PROGRAM MAIN
VAR_INPUT
	// Nostimen tulot
	iElevatorSensor AT %IX1.0: BOOL; // nostimen valoanturi
	iElevatorIsLifted AT %IX1.1: BOOL; // nostin on ajettu ylärajalle
	iElevatorIsDescended AT %IX1.2: BOOL; // nostin on ajettu alarajalle
	iElevatorConveyorRunning AT %IX1.3: BOOL; // nostimen kuljetin pyörii
	
	// Kuljetin 2 tulot
	iConveyor2Sensor AT %IX2.0: BOOL; // Valokenno kuljetin 2 ennen työnnintä
	iPusherPushed AT %IX2.1: BOOL; // Työnnnin on ulkona
	iPusherRetracted AT %IX2.2: BOOL; // Työnnin on sisällä
	iConveyor2Running AT %IX2.3: BOOL; // kuljetin 2 pyörii
	
	// Kuljetin 1 tulot
	iConveyor1Running AT %IX3.0: BOOL; // Kuljetin 1 pyörii
END_VAR

VAR_OUTPUT
	// Kuljetin 1 lähdöt
	qConveyor1 AT %QX0.0: BOOL; // Kuljetin 1 ajo
	
	// Nostimen lähdöt
	qElevatorConveyor AT %QX1.0: BOOL; // Nostimen kuljetin ajo
	qElevatorUp AT %QX1.1: BOOL; // Nostimen nosto ylös
	qElevatorDown AT %QX1.2: BOOL; // Nostimen lasku alas
	
	// Kuljetin 2 lähdöt
	qConveyor2 AT %QX2.0: BOOL; // Kuljetin 2 ajo 
	qPusherPush AT %QX2.1: BOOL; // Työnnin eteen
	qPusherRetract AT %QX2.2: BOOL; // Työnnin taakse
	
	// Laatikon lähtö 
	qBoxShaker AT %QX3.0: BOOL; // Laatikon tärytin
END_VAR

VAR
	ManConveyor1: BOOL; // Kuljetin 1 ajo
	ManElevatorConveyor: BOOL; // Nostimen kuljetin ajo
	ManElevatorUp: BOOL; // Nostimen nosto ylös
	ManElevatorDown: BOOL; // Nostimen lasku alas
	ManConveyor2: BOOL; // Kuljetin 2 ajo 
	ManPusherPush: BOOL; // Työnnin eteen
	ManPusherRetract: BOOL; // Työnnin taakse
	ManBoxShaker: BOOL; // Laatikon tärytin	
	Manual_mode: BOOL;
	Auto_mode: BOOL;
	Lamp: BOOL;
	START: BOOL;
	Seq1: BOOL;
	Seq2: BOOL;
	Seq3: BOOL;
	Seq4: BOOL;
	Seq5: BOOL;
	STOP: BOOL;
END_VAR
VAR // added by the converter: edge detectors and wires of the graphical bodies
    _ft1 : F_TRIG;
    _w1 : BOOL;
END_VAR

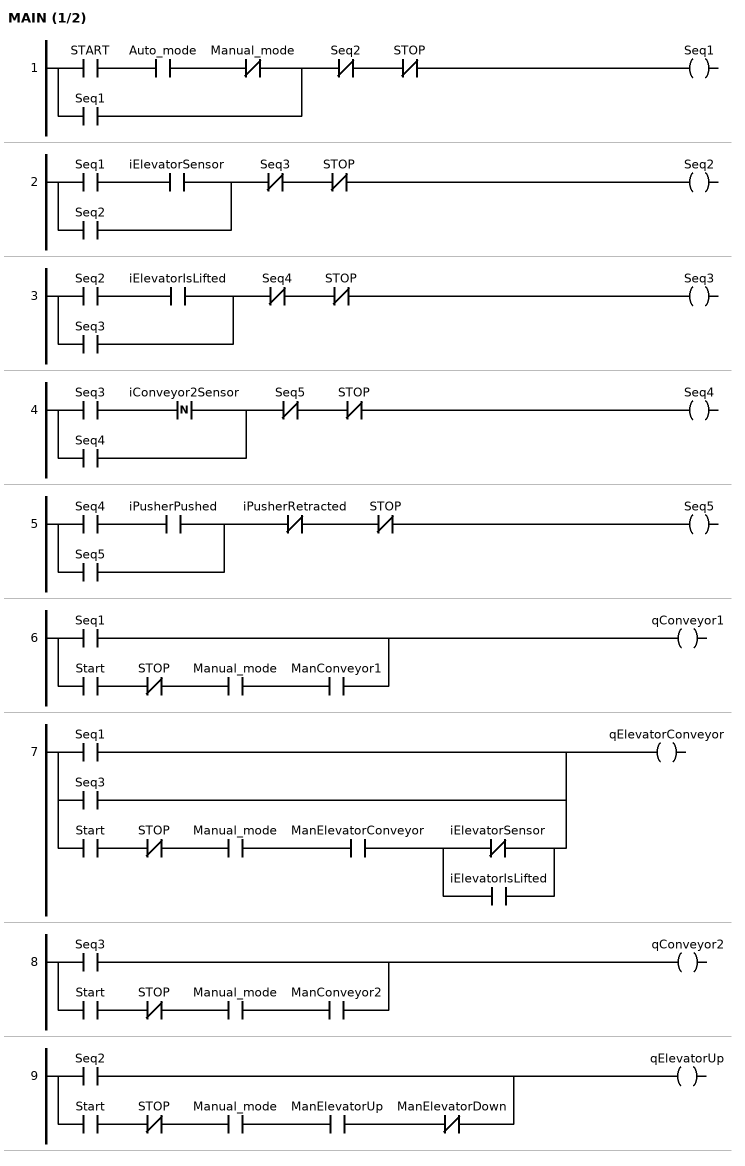
// NETWORK 1
Seq1 := (START AND Auto_mode AND NOT Manual_mode OR Seq1) AND NOT Seq2 AND NOT STOP;

// NETWORK 2
Seq2 := (Seq1 AND iElevatorSensor OR Seq2) AND NOT Seq3 AND NOT STOP;

// NETWORK 3
Seq3 := (Seq2 AND iElevatorIsLifted OR Seq3) AND NOT Seq4 AND NOT STOP;

// NETWORK 4
_ft1(CLK := iConveyor2Sensor);
Seq4 := (Seq3 AND _ft1.Q OR Seq4) AND NOT Seq5 AND NOT STOP;

// NETWORK 5
Seq5 := (Seq4 AND iPusherPushed OR Seq5) AND NOT iPusherRetracted AND NOT STOP;

// NETWORK 6
qConveyor1 := Seq1 OR Start AND NOT STOP AND Manual_mode AND ManConveyor1;

// NETWORK 7
_w1 := Start AND NOT STOP AND Manual_mode AND ManElevatorConveyor;
qElevatorConveyor := Seq1 OR Seq3 OR (_w1 AND NOT iElevatorSensor OR _w1 AND iElevatorIsLifted);

// NETWORK 8
qConveyor2 := Seq3 OR Start AND NOT STOP AND Manual_mode AND ManConveyor2;

// NETWORK 9
qElevatorUp := Seq2 OR Start AND NOT STOP AND Manual_mode AND ManElevatorUp AND NOT ManElevatorDown;

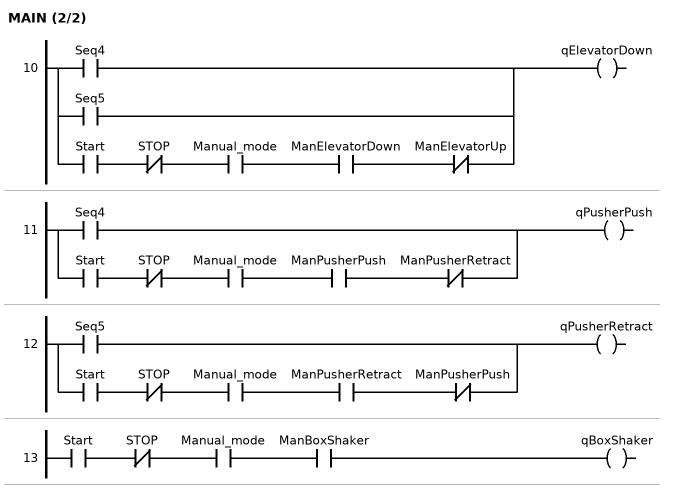
// NETWORK 10
qElevatorDown := Seq4 OR Seq5 OR Start AND NOT STOP AND Manual_mode AND ManElevatorDown AND NOT ManElevatorUp;

// NETWORK 11
qPusherPush := Seq4 OR Start AND NOT STOP AND Manual_mode AND ManPusherPush AND NOT ManPusherRetract;

// NETWORK 12
qPusherRetract := Seq5 OR Start AND NOT STOP AND Manual_mode AND ManPusherRetract AND NOT ManPusherPush;

// NETWORK 13
qBoxShaker := Start AND NOT STOP AND Manual_mode AND ManBoxShaker;

END_PROGRAM

(* stored: Version 1.1.0.1
   POU MAIN: Id {ac9b8f90-2863-4eb9-9843-ccfaa418c12e}, SpecialFunc None *)
